TYPE strBufferHeader :
	STRUCT
		arbyDATA	: ARRAY[1..Sewts_TCP.MAX_BUFFER_SIZE] OF BYTE;
		bJob		: BOOL;		
	END_STRUCT
END_TYPE

(* stored: Version 1.1.0.1, ProductVersion 3.1.4024.12
   DUT strBufferHeader: Id {77127be8-197e-460e-8a10-0b2b0a7588f9} *)
